PROGRAM POU_LAD
VAR
	in_1	: BOOL;
	out_1	: BOOL;
END_VAR

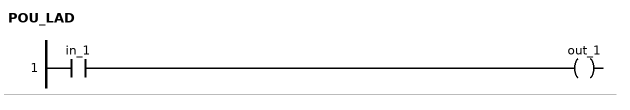
// NETWORK 1
out_1 := in_1;

END_PROGRAM

(* stored: Version 1.1.0.1, ProductVersion 3.1.4024.10
   POU POU_LAD: Id {991d99c1-fee7-4c6b-b8cb-e37041b0a24d}, SpecialFunc None *)
